// Brief: Slave Arm test
FUNCTION_BLOCK PUBLIC FB_SlaveCtrlInstruManualTest EXTENDS FB_SlaveArmCtrlBase
VAR
																
	// final target DH joint position and grip angle
	m_targetDHJntPos:Vec3d;
	m_targetGripAng:LREAL;
	m_targetGripForceLevel :LREAL :=0;
	
	// interploated command joint position and grip angle 
	m_cmdDHJntPos :Vec6d;
	m_cmdDHJntVel :Vec6d;
	m_cmdGripAng:LREAL;

	// last joint position 
	m_lastCmdJntPos :Vec8d ;
	
	// instrument controller
	m_instruController : FB_BasicInstruControl;
	m_usKnifeController : FB_UltrosonicKnifeControl;
	m_instruCmdJntPos,m_instruCmdJntVel : Vec5d;
	m_instruCmdJntTrq :Vec5d;
	
	// OTG
	m_DHJntOTG:ARRAY[1..3] OF FB_secOrdTrajFilter;
	m_gripAngleOTG : FB_secOrdTrajFilter;
	m_maxJntVel:Vec3d:=[3(2.0)];
	m_maxJntAcc:Vec3d:=[3(4.0)];
	
	// instrument tyep
	m_instruType : E_InstrumentType;
	bStart: BOOL;
	iStep: INT;
	fbTon: TON;

	m_maxGripCurrent:LREAL:=350.0;
	m_maxGripCtrlCurrent:LREAL:=540.0;
END_VAR

METHOD PROTECTED calcCmdJntPos : BOOL
VAR_IN_OUT CONSTANT
	i_endoscopePose : ST_Frame;
	i_masterStatus :ST_MasterStatus;
	i_setupStatus: ST_SetupStatus;
	i_slaveArm :FB_SlaveArm;
END_VAR

VAR 
	i:INT :=0;
	errThres :LREAL;
	m_targetDHJntPosLast: Vec3d;
	m_curCmdDHJntPos: Vec3d;
	m_compensationAngleDH: Vec3d;
	m_targetGripAngLast: LREAL;
	m_curCmdAng: LREAL;

END_VAR
// determine target DH joint position and gripper motion
IF GVL_InstruTestUIVars.g_moveToSetPosFlag THEN
	m_targetDHJntPos[1] := GVL_InstruTestUIVars.g_targetRollAng*g_deg2rad;
	m_targetDHJntPos[2] := (GVL_InstruTestUIVars.g_targetPitchAng-90)*g_deg2rad;
	m_targetDHJntPos[3] := GVL_InstruTestUIVars.g_targetYawAng*g_deg2rad;
	IF GVL_InstruTestUIVars.g_targetGripAng>-15 AND GVL_InstruTestUIVars.g_targetGripAng<100  THEN 
		m_targetGripAng := GVL_InstruTestUIVars.g_targetGripAng*g_deg2rad;
		m_targetGripForceLevel:=0;
	ELSIF GVL_InstruTestUIVars.g_targetGripAng<=-15 AND GVL_InstruTestUIVars.g_targetGripAng>=-100 THEN 
		m_targetGripAng := -15*g_deg2rad;
		m_targetGripForceLevel := LIMIT(0, ABS(GVL_InstruTestUIVars.g_targetGripAng), 100);
	ELSIF GVL_InstruTestUIVars.g_targetGripAng<-101 THEN 
		m_targetGripAng := 60 *g_deg2rad;
		m_targetGripForceLevel := LIMIT(-100, 100+GVL_InstruTestUIVars.g_targetGripAng, 0);
	END_IF
ELSIF GVL_InstruTestUIVars.g_gripperOpenFlag THEN
	m_targetGripAng := i_slaveArm.instrument.instruTypeInfo.m_maxGripAngle;
	m_targetGripForceLevel :=0;
ELSIF GVL_InstruTestUIVars.g_gripperCloseFlag THEN
	m_targetGripAng := 0;
	m_targetGripForceLevel :=0;
ELSIF GVL_InstruTestUIVars.g_maxGripForceFlag THEN
	m_targetGripAng := -45*g_deg2rad;
	m_targetGripForceLevel :=100;
END_IF

IF GVL_InstruTestUIVars.m_cycleStart THEN 
	bStart:=TRUE;
	GVL_InstruTestUIVars.m_cycleStart:=FALSE;
END_IF
IF GVL_InstruTestUIVars.m_cycleStop THEN 
	bStart:=FALSE;
	GVL_InstruTestUIVars.m_cycleStop:=FALSE;
END_IF
fbTon(IN:=iStep=10,PT:=T#1S);
IF bStart THEN
	CASE iStep OF 
		0:
			m_targetGripAng := i_slaveArm.instrument.instruTypeInfo.m_maxGripAngle;
			m_targetGripForceLevel :=0;
			iStep:=5;
		5:
		    IF ABS(m_cmdGripAng- m_targetGripAng)< g_jntCtrlAngTolLow THEN
				iStep:=10;
			END_IF
		10:
			IF fbTon.Q THEN
				m_targetGripAng := -90*g_deg2rad;
				m_targetGripForceLevel :=0;
				iStep:=15;
			END_IF
		15:
		    IF ABS(m_cmdGripAng- m_targetGripAng)< g_jntCtrlAngTolLow THEN
				iStep:=0;
			END_IF
	END_CASE
END_IF
// run OTG
FOR i:=1 TO 3  DO
	m_DHJntOTG[i].run(m_targetDHJntPos[i],0.0, o_cmdAcc=>,o_cmdVel=>m_cmdDHJntVel[i],o_cmdPos=> m_cmdDHJntPos[i+3]);
END_FOR
m_gripAngleOTG.run(m_targetGripAng,0.0, o_cmdAcc=>,o_cmdVel=>,o_cmdPos=>m_cmdGripAng);

// calculate target motor joint position from DH joint position
i_slaveArm.instrument.instruIK(m_cmdDHJntPos,m_cmdGripAng, o_jntPos=>m_cmdJntPos);

// command velocity
vecSub(m_cmdJntPos, m_lastCmdJntPos, m_cmdJntVel);
vecSelfMultiNum(m_cmdJntVel, g_slaveArmCtrlFreq);
m_lastCmdJntPos:=m_cmdJntPos;
END_METHOD

// override this function in each exact controller
METHOD PROTECTED calcCmdJntTrq : BOOL
VAR_IN_OUT CONSTANT
	i_endoscopePose : ST_Frame;
	i_masterStatus :ST_MasterStatus;
	i_setupStatus: ST_SetupStatus;
	i_slaveArm :FB_SlaveArm;
END_VAR

VAR 
	nullspaceMat :Mat7d;
	ctrlTrq : Vec7d;
	i : int ;
END_VAR
// set joint torque to zero in default
m_cmdJntTrq := g_zeroVec8d;

// instrument joint control
FOR i:=1 TO 5 DO 
	m_instruCmdJntPos[i]:=m_cmdJntPos[i+3];
	m_instruCmdJntVel[i]:=m_cmdJntVel[i+3];
END_FOR

IF i_slaveArm.instrument.instruType = InstruType_UltrasoundKnifeS OR i_slaveArm.instrument.instruType = InstruType_UltrasoundKnifeU THEN
	m_usKnifeController.run(m_instruCmdJntPos,m_instruCmdJntVel, m_targetGripForceLevel, i_slaveArm, o_cmdJntTrq=>m_instruCmdJntTrq);
ELSE
	m_instruController.run(m_instruCmdJntPos,m_instruCmdJntVel, m_cmdDHJntPos[6], m_cmdDHJntVel[6], m_targetGripForceLevel, i_slaveArm, o_cmdJntTrq=>m_instruCmdJntTrq);
END_IF

FOR i:=1 TO 5 DO
	m_cmdJntTrq[i+3]:=m_instruCmdJntTrq[i];
END_FOR
END_METHOD

METHOD PUBLIC init : BOOL
VAR_IN_OUT CONSTANT
	i_slaveArm	:FB_SlaveArm;
END_VAR
VAR_IN_OUT 
	r_slaveArmCtrlCmd :ST_SlaveArmCtrlCmds;
END_VAR

VAR
	i:int;
END_VAR
SUPER^.Init(i_slaveArm,r_slaveArmCtrlCmd);
m_lastCmdJntPos:=m_cmdJntPos;
m_jntOPMode[1] := DriverOPMode_PosTrq;
m_jntOPMode[2] := DriverOPMode_PosTrq;
m_jntOPMode[3] := DriverOPMode_PosTrq;
m_jntOPMode[4] := DriverOPMode_Trq;
m_jntOPMode[5] := DriverOPMode_Trq;
m_jntOPMode[6] := DriverOPMode_Trq;
m_jntOPMode[7] := DriverOPMode_Trq;
m_jntOPMode[8] := DriverOPMode_Trq;

m_cmdDHJntPos :=i_slaveArm.curDHJntPos;
m_cmdDHJntVel :=g_zeroVec6d;
m_targetGripAng := i_slaveArm.curGripAngle;
m_targetDHJntPos[1] := i_slaveArm.curDHJntPos[4];
m_targetDHJntPos[2] := i_slaveArm.curDHJntPos[5];
m_targetDHJntPos[3] := i_slaveArm.curDHJntPos[6];

// init instrument controller
m_instruController.init(i_slaveArm,m_maxGripCurrent,m_maxGripCtrlCurrent);
m_usKnifeController.init(i_slaveArm);
iStep:=0;
bStart:=FALSE;
IF GVL_InstruTestUIVars.g_rotationAngularVel=0 THEN GVL_InstruTestUIVars.g_rotationAngularVel:=5;END_IF
IF GVL_InstruTestUIVars.g_pitchAngularVel=0 THEN GVL_InstruTestUIVars.g_pitchAngularVel:=5;END_IF
IF GVL_InstruTestUIVars.g_deviationAngularVel=0 THEN GVL_InstruTestUIVars.g_deviationAngularVel:=5;END_IF
IF GVL_InstruTestUIVars.g_rotationAngularAcc=0 THEN GVL_InstruTestUIVars.g_rotationAngularAcc:=30;END_IF
IF GVL_InstruTestUIVars.g_pitchAngularAcc=0 THEN GVL_InstruTestUIVars.g_pitchAngularAcc:=30;END_IF
IF GVL_InstruTestUIVars.g_deviationAngularAcc=0 THEN GVL_InstruTestUIVars.g_deviationAngularAcc:=30;END_IF
FOR i:=1 TO 3  DO
	m_maxJntVel[i]:=5;
	m_maxJntAcc[i]:=30;
	IF GVL_InstruTestUIVars.g_account.actualPermission=2 THEN
		m_maxJntVel[1]:=GVL_InstruTestUIVars.g_rotationAngularVel;
		m_maxJntVel[2]:=GVL_InstruTestUIVars.g_pitchAngularVel;
		m_maxJntVel[3]:=GVL_InstruTestUIVars.g_deviationAngularVel;
		m_maxJntAcc[1]:=GVL_InstruTestUIVars.g_rotationAngularAcc;
		m_maxJntAcc[2]:=GVL_InstruTestUIVars.g_pitchAngularAcc;
		m_maxJntAcc[3]:=GVL_InstruTestUIVars.g_deviationAngularAcc;
	END_IF
END_FOR

FOR i:=1 TO 3  DO
	m_DHJntOTG[i].init(m_cmdDHJntPos[i+3], 0, m_maxJntVel[i], m_maxJntAcc[i], g_slaveArmCtrlCycleTime);
END_FOR

m_gripAngleOTG.init(m_targetGripAng, 0, 2*m_maxJntVel[3], 2*m_maxJntAcc[3], g_slaveArmCtrlCycleTime);
// update commands to arm
copyCmds(r_slaveArmCtrlCmd);
END_METHOD

PROPERTY InstruBacklash : Vec5d
GET
IF m_instruType = InstruType_UltrasoundKnifeS OR m_instruType = InstruType_UltrasoundKnifeU THEN
	instruBacklash := g_zeroVec5d;
ELSE
	instruBacklash := m_instruController.m_jntBacklash;
END_IF
END_GET
END_PROPERTY

END_FUNCTION_BLOCK

(* stored: Version 1.1.0.1, ProductVersion 3.1.4024.11
   POU FB_SlaveCtrlInstruManualTest: Id {dbf632a1-f924-4c4a-9c08-3e3912584188}, SpecialFunc None
   Method calcCmdJntPos: Id {9ac6c1d4-8249-4e40-93a3-6d5814eb3008}
   Method calcCmdJntTrq: Id {672b1be1-2807-47dd-8f1d-525fb978a27b}
   Method init: Id {406632cf-8059-46ab-b0c2-acbe734ef5ab}
   Property InstruBacklash: Id {b8a24ea9-b582-4c33-9d96-935e62686f4d}
   Get Get: Id {b3292599-741b-4cc2-b2a4-345b2cfdea2c} *)
